{attribute 'GeneratedUsingTerminal: EL5001-0000-1017'}
{attribute addProperty BoxType "EL5001-0000-1017"}
{attribute addProperty Description "EL5001 1Ch. SSI Encoder"}
{attribute addProperty Physics "KK"}
{attribute addProperty Id "SSI_InputsAT %I*SSI_Inputs_0E3D8E3310WcStateAT %I*WcState_9091E0EB2InfoDataAT %I*InfoData_32EB74EA10"}
{attribute addProperty CRC "187224199"}
{attribute addProperty Size "22"}
TYPE EL5001_0B28D087 EXTENDS EtcSlaveTerminalBase_947E5A46 :
STRUCT
	{attribute addProperty Name "SSI_Inputs"}
	SSI_Inputs : SSI_Inputs_0E3D8E33;
	{attribute addProperty Name "WcState"}
	WcState : WcState_9091E0EB;
	{attribute addProperty Name "InfoData"}
	InfoData : InfoData_32EB74EA;
END_STRUCT
END_TYPE

(* stored: Version 1.2.0.0, ProductVersion 3.1.4024.9
   DUT EL5001_0B28D087: Id {8a8456be-7a89-4f56-b131-dea0ccfd11a0} *)
